# EPICS StreamDevice protocol: EthercatMCApp/Db/UTCtime.proto
# Protocol file to get the (local)nUTC time from the motion controller
#
##################################################
# General Settings
##################################################

Terminator = LF;
ReplyTimeout = 1000;

###################################################
# Get functions
###################################################
getUTCtime {
   out "ADSPORT=852/Main.sTime?;";
   in "%23c;";
}
